INTERFACE I_AlarmVisitor

METHOD VisitError
VAR_INPUT
	VisitingError : I_Alarm;
END_VAR
END_METHOD

END_INTERFACE

(* stored: Version 1.1.0.1, ProductVersion 3.1.4024.12
   Itf I_AlarmVisitor: Id {41a9b258-2373-0f62-3efc-013219d20622}
   Method VisitError: Id {ef0ab7c6-07b4-06c4-07b2-8969432c5267} *)
